Universal Robots URScript: SUB_7002.script

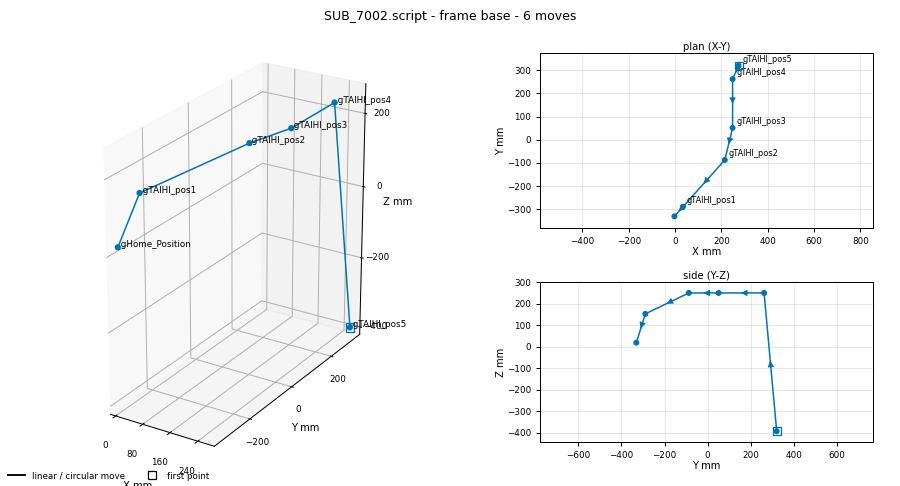
[picture p0: tool path of SUB_7002.script in frame base, 6 of 6 moves have a stored position in this frame; points joined in program order, loops and branches not executed]
def SUB_7002():
  global _hidden_verificationVariable=0
  step_count_d413a972_fa5a_4f2e_8905_9a2c59b730f0 = 0.0
  thread Step_Counter_Thread_81efb043_53a0_42e3_b210_04cebb1d3d18():
    while (True):
      step_count_d413a972_fa5a_4f2e_8905_9a2c59b730f0 = step_count_d413a972_fa5a_4f2e_8905_9a2c59b730f0 + 1.0
      sync()
    end
  end
  run Step_Counter_Thread_81efb043_53a0_42e3_b210_04cebb1d3d18()
  set_gravity([0.0, 0.0, 9.82])
  set_tcp(p[0.0,0.06,0.45,0.0,0.0,0.0])
  set_standard_analog_input_domain(0, 1)
  set_standard_analog_input_domain(1, 1)
  set_tool_analog_input_domain(0, 1)
  set_tool_analog_input_domain(1, 1)
  set_analog_outputdomain(0, 0)
  set_analog_outputdomain(1, 0)
  set_input_actions_to_default()
  set_runstate_gp_boolean_output_to_value(0, 3)
  set_tool_communication(False, 115200, 0, 1, 1.5, 3.5)
  set_tool_output_mode(0)
  set_tool_digital_output_mode(0, 1)
  set_tool_digital_output_mode(1, 1)
  set_tool_voltage(0)
  set_target_payload(0.100000, [0.135000, 0.000000, 0.225000], [10.000000, 10.000000, 10.000000, 0.000000, 0.000000, 0.000000])
  set_safety_mode_transition_hardness(1)
  global isReCapt=False
  global Bucket_Z=[0, 0.7]
  global DistPillar=-305.86292
  global CandCnt=1
  global lr=1
  global ReCaptZ=0.05
  global forceval=p[0, 0, 0, 0, 0, 0]
  global CaptDepth=[0.26, 0.24, 0]
  global port=3000
  global isOnlyF=True
  global retX2=p[-0.01249, 0.23197, 0.03388, -0.03334, 0.03134, -1.47265]
  global socket_timeout=120
  global isSkipP=False
  global curpos=p[0, 0, 0, 0, 0, 0]
  global host="192.168.1.2"
  global is_popup=False
  global CaptZOffset=0
  global isGoHome=True
  global i_pos2=p[-0.68095, 0.14083, -0.02528, 1.97677, 2.1368, 0.30928]
  global i_pos1=p[-0.68039, 0.14096, -0.02512, 1.97601, 2.13656, 0.31051]
  global pBucket=[p[0.76533, 0.44669, 0.35721, 0, 0, -1.54409], p[-0.77489, -0.51021, 0.35436, 0, 0, 1.63138], p[0, 0, 0, 0, 0, 0]]
  global CaptStepZ=0.08
  global CaptIndex=[0, 0, 0]
  global CaptStepX=0.432
  global pBucketM=p[-0.80141, -0.42542, 0.2879, 0, 0, 1.55713]
  global socket_name="vt"
  global rovi_err=0
  global SubPrgResult=100
  global CurrPos=p[0.03109, -0.36281, 0.46695, -0.00903, -3.12835, 0.092]
  global CurrPos_p=p[0.026, -0.32934, 0.01423, -0.00903, -3.12835, 0.092]
  global ForceStartZ=0.43617
  global CutOffZ=0.08
  global HomeDistTh=0.05
  global RBDistTh=0.05
  global RBRadiusTh=0.3
  global RBXTh=[-0.5, 0.5]
  global RBYTh=[-0.8, 1]
  global RBZTh=[-0.1, 0.1]
  global Sub3100_ZMax=0.74
  global ForceStartX=-0.90368
  global Sub3100_aRot=0.2
  global Sub3100_d=0.3
  global Sub3100_Option=1
  global Sub3100_a=0.2
  global Sub3100_XdV=0.1
  global Sub3100_XdRot=8
  global ZoneDistTh=0.05
  global ZoneRadiusTh=0.3
  global ZoneXTh=[-0.5, 0.5]
  global ZoneYTh=[-0.8, 1]
  global ZoneZTh=[-0.1, 0.1]
  global BucketWidth=0.95
  global ZoneBucketGap=0
  global ZoneHomeX=0.2
  global UnloadZ=0.05
  global CaptPos=p[0.4274, -0.37367, -0.0279, 3.13247, 0.05506, 0.01735]
  global BucketUpperPos=p[0.4274, -0.37367, -0.0279, 3.13247, 0.05506, 0.01735]
  global Sub3100_GPII18=1
  global Zone6ThX=0.1
  global Zone6ThY=0.05
  global Bucket=p[0.32604,0.49174,0.0,-1.882900624652718E-5,2.8304179127934987E-5,-1.593185305749222]
  global BucketM=p[0.32604,0.49174,0.0,2.2353980716304163E-16,-3.5868426080024975E-16,-1.5931853071795856]
  global CaptPoint_C=p[-0.4219337985373468,-0.003168602281063755,0.26,-2.1962364319979395,-2.2439316084554193,-0.02184884826814999]
  global CaptPoint_C2=p[0.32796661698047924,-0.010768520544682924,0.01931625281283378,2.2288103429550152,-2.213636886217198,8.598462540813273E-5]
  global CaptPoint_L=p[-0.42193494849366175,-0.2,0.26,-2.1962086037526625,-2.2438965822622805,-0.02199725151111115]
  global CaptPoint_L2=p[0.327894307417917,-0.010799940826224014,0.01928712668893995,2.087717047309385,-2.0736781215133306,0.27365839887453103]
  global CaptPoint_R=p[-0.4219551896101372,0.3,0.26,-2.1960823751563487,-2.2439541235147065,-0.021863042557804555]
  global CaptPoint_R2=p[0.327926308680866,-0.010795166414457658,0.019300245403843563,-2.1186306375223185,2.1040550557443427,0.22023197678473694]
  global Capt_1BK_L=p[-0.4574214308482636,-0.48457071473611046,0.3504487959434708,-2.1962343446504526,-2.243967222238911,-0.021809195357489434]
  global Capt_1BK_R=p[-0.4574597285646511,0.4755214243904677,0.35039311859649847,-2.196330286580149,-2.2438949166739053,-0.021738621025254933]
  global Capt_1BK_pos1=p[-0.4218793038724447,-0.003154429464978058,0.2915499891144615,-2.1963422029204875,-2.2438663520270015,-0.02197160668673838]
  global Capt_1BK_pos2=p[-0.42187829024618434,-0.0031710253373066375,0.29156503858953065,-2.196324918349679,-2.2439040699490773,-0.021928444416953782]
  global Capt_2BK_L=p[0.42186661528427194,0.4254738068040517,0.35042275762909847,2.239156309475874,-2.1837044610999294,0.002643817066643282]
  global Capt_2BK_R=p[0.4218208572756906,-0.5427676723257963,0.350372239919558,2.2392697861179327,-2.183553596194912,0.002410470905346486]
  global Capt_2BK_pos1=p[0.42193501458435656,0.004742683868356356,0.35045865974037793,2.2391012408536453,-2.1839704655717003,0.002677867056024068]
  global Capt_2BK_pos2=p[0.421903984494575,0.004707988774967922,0.35045218900915065,2.239114367170047,-2.183895515396197,0.002684056681074047]
  global Capt_GD_M=p[-0.004053197679954899,-0.25261725691632436,-0.01970497430780127,0.0332779454553888,-3.140179196376707,-0.0034093680964018282]
  global HomePointL=p[-0.36789,-0.5117344641471838,0.78,-0.6278857271586024,3.0680899128661667,-8.649957362498864E-4]
  global PickPos=p[0.10830682331105715,-1.3709505888096256,-0.18404188875951455,-0.00622194000158997,2.880236948927292,-0.00383636509397631]
  global Solve=p[-0.00368,-0.0021000000000000003,0.25739999999999996,0.0,0.0,0.0]
  global TCP3100TL=p[0.0,0.06,0.535,1.8939999999999997,0.0,0.0]
  global TEST=p[0.1,0.0,0.2,0.0,0.0,0.0]
  global UF=p[0.0,0.0,0.0,0.0,0.0,0.0]
  global g1CV_1_M=p[0.29093319989156785,-0.9405344885124904,-0.08686754932079166,1.9884186265311852,2.2323374792844253,0.1524643645929425]
  global g1CV_posL1=p[0.05028133628211688,-0.4526481033729615,0.1221845548632916,-2.213335080948508,-2.1937561336067057,-0.3280056759040735]
  global g1CV_posR1=p[0.03743870476062511,-0.53119407812668,0.11301901343688614,2.073418671558482,2.153257467049566,0.11656306439039889]
  global g1GD_pos1=p[0.06841781024889843,-0.5456037307108855,0.367146167315866,2.4108578981103275,1.7957834606331096,0.12544942012730473]
  global g1GD_pos2=p[0.06838772140470781,-0.5455736997413498,0.3671086150887749,2.4109085778803876,1.795859110102632,0.12543092350975993]
  global g1GD_pos3=p[-0.12994435620230207,-0.4431007958053758,0.36202773375526215,2.579773746707185,1.5871477668617076,0.08382931926093913]
  global g1GD_pos4=p[-0.19950049720405605,-0.020433345237594124,0.36213807486671723,2.098425945606484,2.2067222807383033,0.12502137451358736]
  global g1GD_pos5=p[-0.6594126711541819,-0.02045920875309877,0.36212219059276163,2.0984573928915715,2.2065752443497044,0.12515745843348272]
  global g1GD_posL1=p[-0.08276848269606216,-0.3996147100031649,0.1488453551331823,2.286527078917204,1.8420745504477611,0.33698451773695576]
  global g1GD_posL2=p[-0.3253977027403738,-0.3024804624281039,0.16332814085945146,2.72312820760317,0.9631021078169197,0.32447452035226126]
  global g1GD_posL3=p[-0.6791033397183219,0.06787475590683856,0.16337212788108813,2.1383125299263996,2.086116032377724,0.4536080263755059]
  global g1GD_posR1=p[-0.09893370538053747,-0.4999608954567234,0.14329885217724153,2.43311852414254,1.4238397520832589,0.08559216753941556]
  global g1GD_posR2=p[-0.3729565201882258,-0.3752983669473301,0.143299052800563,2.6951655216297596,0.8130506811102118,-0.02387549506099888]
  global g1GD_posR3=p[-0.7385929502572233,-0.029472684480355026,0.1499650660949685,2.0484522752014467,1.9493695704119496,0.18368227556562683]
  global g2CV_1_M=p[0.26887505416660307,-0.9603120922602274,-0.007666051543921415,2.1502738513797834,2.1807891159519985,0.05286430186756905]
  global g2CV_posL1=p[0.3409386496330911,-0.4656338066361442,0.1250074988128972,2.209372209162659,2.1945371304665926,0.3160714960040194]
  global g2CV_posR1=p[0.3400736278759575,-0.531334269888987,0.1183415684753657,2.07314649492589,2.1532617466521136,0.11638666128062146]
  global g2GD_pos1=p[0.3390086633742754,-0.5203839341398588,0.22258,2.022696172282159,2.259224887850344,0.09811005079237367]
  global g2GD_pos2=p[0.4140891885236144,0.14850105084950693,0.1582916370575993,-0.10302503203970696,3.1008909166713883,0.18748967846962497]
  global g2GD_pos3=p[0.32377086541216454,-0.01023215987367155,0.15821240334102793,2.279746475463588,-2.06129961332614,-0.16578334012307952]
  global g2GD_pos4=p[0.5908983921852361,0.05403340620320105,0.22256644303459816,2.1622925298497893,-2.1689699585948934,-0.13856866383637143]
  global g2GD_pos5=p[0.3170888000905397,0.12187007662842038,0.22197674485563323,0.8377606158495782,-3.0022727604914152,-0.17086710591731175]
  global gCV_11_M=p[0.2952490857586,-0.9656006017777,-0.0031848736745567763,2.0722728991542883,1.9962782396866086,0.36470882731217735]
  global gCV_12_M=p[0.33130761172890943,-0.9656131260212175,-0.003202101878453989,2.0724239607469284,1.9962431566902565,0.3645969752142286]
  global gCV_13_M=p[0.36489346066019257,-0.9655807239160527,0.06876536645596665,2.072464232199882,1.9963052684095466,0.3646153924747167]
  global gCV_14=p[0.35645641620611146,-0.8914305774826713,-0.17737239800677018,2.1506886654737776,2.1461343800624295,0.40986447399780934]
  global gCV_15=p[0.4370373250739419,-0.891408661166693,-0.1773997714481486,2.1507483614991094,2.1461657601704176,0.40983132876462236]
  global gCV_16=p[0.4597123429384979,-0.8913837618729653,-0.03599504377258328,2.1506156333226136,2.1462305295546718,0.4099109158136618]
  global gCV_17=p[0.037528034463104695,-0.6904892259828748,-0.12243237639232962,-0.12012393052395552,2.832430475095037,0.48967048060305135]
  global gCV_18=p[0.03600103065313248,-0.6368623043127666,-0.12241687036449483,-0.12010351348807546,2.832474314609516,0.48970816626953567]
  global gCV_2_M=p[0.26884116022244575,-0.9602965195051723,0.05955583488779087,2.150403327161483,2.180756105286659,0.05289689171405361]
  global gCV_3_M=p[0.29099390607376485,-0.6570558385379063,0.0722153583041818,1.9884242634571576,2.2321538498123994,0.15249643504377583]
  global gCV_5=p[0.045776199142861046,-0.9791473230816141,0.8415069045351792,2.0229894037377316,2.080009888728606,0.35618099403901887]
  global gCV_pos5=p[0.3400172856834047,-0.9722754606605235,-0.18287928563575456,2.073394561413637,2.1531827558666565,0.11639000988241816]
  global gGD_100_1LM=p[0.04146780808756359,-0.6870904124925177,-0.1232943093634104,-0.006305250057386166,-2.863965809273829,-0.5082528300185785]
  global gGD_1_LM=p[0.020434109115523666,-0.7173924052060343,-0.08811,-0.04183287991373406,2.838581017021502,0.4853906791299838]
  global gGD_1_M=p[0.02544173067907144,-0.7152638990611948,-0.08715105875448259,0.03146811630679845,3.078203630151714,0.5317053337229012]
  global gGD_1_MM=p[0.025400458185448213,-0.6216049814301073,0.010176266954312452,0.03131467408099384,3.0782064649052026,0.5315951524792814]
  global gGD_1_RM=p[0.031217318880483708,-0.7147335545146203,-0.08957999999999999,-0.08489904435139688,-2.8488123547477313,-0.48120690485983686]
  global gGD_200_2LM=p[0.04175812558137225,-0.6358261219893102,-0.12285474020423298,-0.006257718193554584,-2.863964784148567,-0.5084621939645108]
  global gGD_2_LM=p[0.02018390025483749,-0.6687426063994015,-0.08718000000000001,-0.041835187515792314,2.8386379488451055,0.485489484053296]
  global gGD_2_M=p[0.025409431193568414,-0.6711183508441593,-0.08720488631611445,0.03149312968575293,3.07816411505092,0.5318561240593018]
  global gGD_2_RM=p[0.031210703641741028,-0.6710692701219645,-0.08952,-0.08481788616135903,-2.8489140382691294,-0.48104729490717946]
  global gGD_300_3LM=p[0.04182050265947469,-0.6066076810742604,-0.03602288107395374,-0.006290924000441408,-2.8640915241774816,-0.5083501301248439]
  global gGD_3_LM=p[0.020461334165751577,-0.6291141807342636,0.0118532658633555,-0.04183776139390022,2.838559087651966,0.48540926433742404]
  global gGD_3_M=p[0.02533516482015475,-0.6215615348897825,0.010200828403046092,0.031513364919278905,3.078253870709586,0.5317609336513714]
  global gGD_3_RM=p[0.031260390466643626,-0.6224758015041261,0.012117368031848541,-0.08473182226111171,-2.848909743557149,-0.4810787915420777]
  global gGD_400_1RM=p[0.03765496539143813,-0.6905733748742057,-0.12240702670509729,-0.12009639012349203,2.8324503628258273,0.48945657912051843]
  global gGD_4_LM=p[-0.1344797585014677,-0.6291858144255682,0.01186447051560996,-0.04187273583495941,2.8385192271564894,0.48521441537128857]
  global gGD_4_RM=p[0.17738270383844643,-0.622513694547901,0.01211517030876813,-0.08466921567219163,-2.848954628800666,-0.48095852370908404]
  global gGD_500_2RM=p[0.0364038044475721,-0.6361408639594927,-0.1228896102948493,-0.12001814478849077,2.8324363686538967,0.4895422385690364]
  global gGD_600_3RM=p[0.03597788557419286,-0.6039591135870097,-0.03251312847845622,-0.12016380804709932,2.832584395249392,0.4895204315491753]
  global gGD_M_20=p[0.03524102305764369,-0.704963855446233,-0.12310321086399345,-0.05961230604660993,3.0873078767639504,0.5414261100507907]
  global gGD_M_30=p[0.03527181411394771,-0.6949613298581867,-0.12309199448652725,-0.05962447301074729,3.087287038166274,0.5412100180254447]
  global gGD_M_40=p[0.035236425258241534,-0.6834410208824955,-0.12309554834290798,-0.05953064339288712,3.087315110349415,0.5412921265180426]
  global gHome_Position=p[-0.0028466672127084513,-0.33076167646145177,0.018757637154973972,0.022264309958481422,3.141485447328174,-2.928857653237729E-4]
  global gTAIHI_pos1=p[0.03440188678018217,-0.2890699997284216,0.1524459153418134,0.03555253805738487,3.139753660134215,-0.0072926847345475936]
  global gTAIHI_pos2=p[0.21480420508123035,-0.08727040094693181,0.2494872417251085,0.0993881044708114,3.130169265768029,-0.041005976873124614]
  global gTAIHI_pos3=p[0.24842855789766727,0.05125360387123426,0.24954489042226397,-1.3393932107301392,2.8188336257431876,-0.029365966672838972]
  global gTAIHI_pos4=p[0.2484136724826812,0.2619974016830966,0.249555843497129,-2.9133089622066395,1.099075078448136,0.0012284823840295143]
  global gTAIHI_pos5=p[0.2742702426594438,0.32043482129403583,-0.39188788327742546,-3.110801532722998,0.17164161774330408,0.0023707125334252723]
  rtde_set_watchdog("speed_slider_mask", 10.0, "ignore")
  # begin: URCap Installation Node
  #   Source: Ethernet/IP I/O Monitor URCap, 1.0.0,
  #   Type: Ethernet/IP I/O Monitor
  conn = rpc_factory("xmlrpc", "http://127.0.0.1:" + to_str(61101) + "/RPC2")

  def show_monitor():
    return conn.eip_monitor.show()
  end
  # end: URCap Installation Node
  while (True):
    $ 2 "ロボットプログラム"
    $ 3 "設定"
    set_tcp(p[0.0,0.06,0.45,0.0,0.0,0.0])
    $ 4 "荷重の設定: k10"
    set_target_payload(0.100000, [0.135000, 0.000000, 0.225000], [10.000000, 10.000000, 10.000000, 0.000000, 0.000000, 0.000000])
    $ 5 "MoveL"
    $ 6 "gTAIHI_pos5" "breakAfter"
    movel(gTAIHI_pos5, a=0.07, v=0.12)
    $ 7 "gTAIHI_pos4" "breakAfter"
    movel(gTAIHI_pos4, a=0.07, v=0.12)
    $ 8 "gTAIHI_pos3" "breakAfter"
    movel(gTAIHI_pos3, a=0.07, v=0.12)
    $ 9 "gTAIHI_pos2" "breakAfter"
    movel(gTAIHI_pos2, a=0.07, v=0.12)
    $ 10 "gTAIHI_pos1" "breakAfter"
    movel(gTAIHI_pos1, a=0.07, v=0.12)
    $ 11 "gHome_Position" "breakAfter"
    movel(gHome_Position, a=0.07, v=0.12)
    $ 12 "停止"
    halt
  end
end
